{attribute 'c++_compatible'}
FUNCTION_BLOCK FB_DoWork EXTENDS TcBaseModuleRegistered IMPLEMENTS I_DoWork

METHOD FB_reinit : BOOL
SUPER^.FB_reinit();
END_METHOD

{attribute 'TcTypeSystem'}
{attribute 'c++_compatible'}
{attribute 'minimal_input_size' := '4'}
{attribute 'pack_mode' := '4'}
METHOD M_Increment : Global.HRESULT
VAR_INST
	fbCrititcalSection : FB_IecCriticalSection;
	fbRTMon_LogMark	   : FB_RTMon_LogMark;
	_counter		   : UDINT;	
END_VAR
IF fbCrititcalSection.Enter() THEN
	(* start of critical section *)
	fbRTMon_LogMark.LogStart(0, 0);
	_counter := _counter + 1;
	F_ConsumeTime(100);
	M_Increment := S_OK;
	fbRTMon_LogMark.LogStop(0, 0);

	(* end of critical section *)
	fbCrititcalSection.Leave();
END_IF
END_METHOD

{attribute 'minimal_input_size' := '4'}
{attribute 'pack_mode' := '4'}
{attribute 'c++_compatible'}
METHOD TcQueryInterface : Tc3_Module.HRESULT
VAR_INPUT
	iid	   : REFERENCE TO Tc3_Module.IID;
	pipItf : POINTER TO Tc3_Module.PVOID;
END_VAR

VAR
	ipDoWork : I_DoWork;
END_VAR
IF GuidsEqual(ADR(iid), ADR(TC_GLOBAL_IID_LIST.IID_I_DoWork)) THEN
	ipDoWork := THIS^; // cast to interface pointer
	pipItf^ := ITCUNKNOWN_TO_PVOID(ipDoWork);
	TcAddRef();
	TcQueryInterface := S_OK;
ELSE
	TcQueryInterface := SUPER^.TcQueryInterface(iid, pipItf);
END_IF
END_METHOD

END_FUNCTION_BLOCK

(* stored: Version 1.1.0.1, ProductVersion 3.1.4026.18
   POU FB_DoWork: Id {2ab00ae1-5d1d-4c1b-b03f-8fbf1ff0b8b3}, SpecialFunc None
   Method FB_reinit: Id {9053b03d-8ede-4a48-b24f-aff7895ba10c}
   Method M_Increment: Id {f67746c2-42d3-45f0-81a3-8096efda097c}
   Method TcQueryInterface: Id {7ae69c2f-9bc2-4d19-b54e-9c7ca1339714} *)
